(*
SPDX-FileCopyrightText: © 2026 Oleksandr Tiutyk <trofimich@gmail.com>
SPDX-License-Identifier: MIT
License: https://opensource.org/license/mit
*)

(*!
<summary>Reports an operation that requires an element in an empty collection.</summary>
<description>
The caller detects the condition; this exception does not inspect or modify the collection or destination.
Uses the GeneralException task-local cycle lifetime and throw rules.
</description>
*)
INTERFACE ICollectionEmptyException EXTENDS IGeneralException

(*!
<summary>Builds the diagnostic and raises this exception through GeneralException.</summary>
<description>
Copies the supplied diagnostic data, sets error code to zero and supplies no inner exception. Call only in a
cyclic task, not during FB_init. The caller must already have detected the reported condition.
</description>
<param name="collectionName">Collection name used in the diagnostic.</param>
*)
METHOD Throw
VAR_INPUT
	sourceNamespaceName : STRING;
	sourceClassName : STRING;
	sourcePOUName : STRING;
	sourcePosition : STRING;
	collectionName : WSTRING;
END_VAR
END_METHOD

END_INTERFACE

(* stored: Version 1.1.0.1
   Itf ICollectionEmptyException: Id {60fb87e6-238c-4a7d-9087-bc4ff389d5a3}
   Method Throw: Id {77e34b25-d199-4c45-8866-245dc5f50505} *)
